TYPE ST_Fenster_Steuerung :
STRUCT
	Freigabe			: ST_Steuerung_auto_manu_BOOL;
	Freigabe_Deakt		: ST_Steuerung_auto_manu_BOOL;
	Fenster_AUF			: ST_Steuerung_auto_manu_BOOL;
	Fenster_ZU			: ST_Steuerung_auto_manu_BOOL;
	Quittierung			: BOOL;

END_STRUCT
END_TYPE

(* stored: Version 1.1.0.1, ProductVersion 3.1.4024.9
   DUT ST_Fenster_Steuerung: Id {28ec8b88-a0e3-4d7a-865f-cfc3fe5e51e0} *)
